// TIA Portal project "Food_Production_Automation" (V17)

(* hardware
DEVICE "HMI_1"  KTP700 Basic PN
   slot 0: "HMI_1"  KTP700 Basic PN  6AV2 123-2GB03-0AX0  17.0.0.0
   slot 1: "HMI_RT_1"  KTP700 Basic PN  6AV2 123-2GB03-0AX0  17.0.0.0
   slot 5: "HMI_1.IE_CP_1"  PROFINET Interface  17.0.0.0
      slot 1: "PROFINET Interface_1"  PROFINET Interface
         slot 1: "Port_1"  Port
DEVICE "S7-1200 station_1"  S7-1200 Station
   slot 0: "Rack_0"  S7-1200 Rack  Rack  V1.0
   slot 1: "PLC_1"  CPU 1215C DC/DC/DC  6ES7 215-1AG40-0XB0  V4.5
   slot 2: "AI 4xRTD_1"  SM 1231 AI4 x RTD  6ES7 231-5PD32-0XB0  V2.0
*)

// ===== PLC "PLC_1"  CPU 1215C DC/DC/DC =====

VAR_GLOBAL   // PLC tag table "Default tag table"
   "Tank 1 Desired Temperature" AT %MD10 : Real;
   "Tank 2 Desired Temperature" AT %MD14 : Real;
   "Tank 1 PT100 Raw" AT %IW96 : Int;
   "Tank 1 PT100 Real" AT %MD18 : Real;
   "Tank 1 Current Temperature" AT %MD22 : Real;
   "Tank 2 PT100" AT %IW98 : Int;
   "Tank 2 PT100 Real" AT %MD26 : Real;
   "Tank 2 Current Temperature" AT %MD30 : Real;
   "HMI Start Stop Button" AT %M34.0 : Bool;
   "Heater 1" AT %Q0.0 : Bool;
   "Heater 2" AT %Q0.1 : Bool;
END_VAR

ORGANIZATION_BLOCK "Main"   // OB1, LAD, ProgramCycle
TITLE = "Main Program Sweep (Cycle)"
{ S7_Optimized_Access := 'TRUE' }
VERSION : 0.1
   VAR_INPUT
      Initial_Call : Bool;   // Initial call of this OB
      Remanence : Bool;   // =True, if remanent data are available
   END_VAR
BEGIN

REGION Network 1
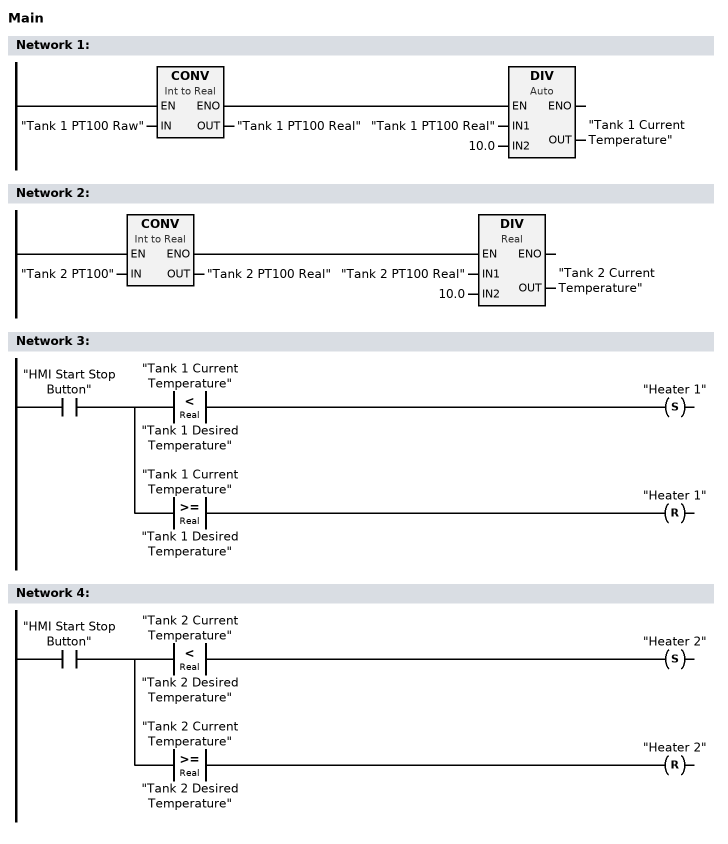
   RUNG wire#powerrail
      { S7_Templates := "[SrcType := Int, DestType := Real]" } Convert(in := "Tank 1 PT100 Raw", out => "Tank 1 PT100 Real")
      Div(in1 := "Tank 1 PT100 Real", in2 := 10.0, out => "Tank 1 Current Temperature")
   END_RUNG
   // the same network as SCL:
   "Tank 1 PT100 Real" := INT_TO_REAL("Tank 1 PT100 Raw");
   "Tank 1 Current Temperature" := "Tank 1 PT100 Real" / 10.0;
END_REGION

REGION Network 2
   RUNG wire#powerrail
      { S7_Templates := "[SrcType := Int, DestType := Real]" } Convert(in := "Tank 2 PT100", out => "Tank 2 PT100 Real")
      { S7_Templates := "SrcType := Real" } Div(in1 := "Tank 2 PT100 Real", in2 := 10.0, out => "Tank 2 Current Temperature")
   END_RUNG
   // the same network as SCL:
   "Tank 2 PT100 Real" := INT_TO_REAL("Tank 2 PT100");
   "Tank 2 Current Temperature" := "Tank 2 PT100 Real" / 10.0;
END_REGION

REGION Network 3
   RUNG wire#powerrail
      Contact( "HMI Start Stop Button" )
      wire#w1
      { S7_Templates := "SrcType := Real" } LT_Contact(in1 := "Tank 1 Current Temperature", in2 := "Tank 1 Desired Temperature")
      S_Coil( "Heater 1" )
   END_RUNG
   RUNG wire#w1
      { S7_Templates := "SrcType := Real" } GE_Contact(in1 := "Tank 1 Current Temperature", in2 := "Tank 1 Desired Temperature")
      R_Coil( "Heater 1" )
   END_RUNG
   // the same network as SCL:
   IF "HMI Start Stop Button" AND ("Tank 1 Current Temperature" < "Tank 1 Desired Temperature") THEN
       "Heater 1" := TRUE;
   END_IF;
   IF "HMI Start Stop Button" AND ("Tank 1 Current Temperature" >= "Tank 1 Desired Temperature") THEN
       "Heater 1" := FALSE;
   END_IF;
END_REGION

REGION Network 4
   RUNG wire#powerrail
      Contact( "HMI Start Stop Button" )
      wire#w1
      { S7_Templates := "SrcType := Real" } LT_Contact(in1 := "Tank 2 Current Temperature", in2 := "Tank 2 Desired Temperature")
      S_Coil( "Heater 2" )
   END_RUNG
   RUNG wire#w1
      { S7_Templates := "SrcType := Real" } GE_Contact(in1 := "Tank 2 Current Temperature", in2 := "Tank 2 Desired Temperature")
      R_Coil( "Heater 2" )
   END_RUNG
   // the same network as SCL:
   IF "HMI Start Stop Button" AND ("Tank 2 Current Temperature" < "Tank 2 Desired Temperature") THEN
       "Heater 2" := TRUE;
   END_IF;
   IF "HMI Start Stop Button" AND ("Tank 2 Current Temperature" >= "Tank 2 Desired Temperature") THEN
       "Heater 2" := FALSE;
   END_IF;
END_REGION
END_ORGANIZATION_BLOCK

(* ===== HMI "HMI_RT_1" =====
system functions are stored by id; their names below are inferred from use
connection "HMI_Connection_1": ETHERNET, SMART_S7_1200_OMS

HMI tags "Default tag table"
   "Tank 1 Desired Temperature" : Real = PLC "Tank 1 Desired Temperature" AT %MD10, 1 s
   "Tank 2 Desired Temperature" : Real = PLC "Tank 2 Desired Temperature" AT %MD14, 1 s
   "Tank 1 Current Temperature" : Real = PLC "Tank 1 Current Temperature" AT %MD22, 1 s
   "Tank 2 Current Temperature" : Real = PLC "Tank 2 Current Temperature" AT %MD30, 1 s
   "Heater 1" : Bool = PLC "Heater 1" AT %Q0.0, 1 s
   "Heater 2" : Bool = PLC "Heater 2" AT %Q0.1, 1 s
   "HMI Start Stop Button" : Bool = PLC "HMI Start Stop Button" AT %M34.0, 1 s

recipe "Recipe_1": Tank 1 Desired Temperature <- "Tank 1 Desired Temperature", Tank 2 Desired Temperature <- "Tank 2 Desired Temperature"

screen "Root screen" 800x480, template "Template_1"
   TextField "Text field_1" at 194,5 size 408x32; Text 'FOOD PRODUCTION AUTOMATION'
   GraphicView "Graphic view_3" at 84,252 size 87x48; Picture "Graphic_3"
   GraphicView "Graphic view_2" at 24,123 size 114x199; Picture "Graphic_2"
   GraphicView "Graphic view_1" at 254,252 size 87x48; Picture "Graphic_3"
   GraphicView "Graphic view_4" at 194,123 size 114x199; Picture "Graphic_2"
   GraphicView "Graphic view_5" at 48,156 size 66x67; Picture "Graphic_4"
   GraphicView "Graphic view_6" at 217,156 size 66x67; Picture "Graphic_4"
   Rectangle "Rectangle_1" at 64,240 size 30x30
      Appearance <- "Heater 1"
   Rectangle "Rectangle_2" at 235,240 size 30x30
      Appearance <- "Heater 2"
   TextField "Text field_2" at 49,294 size 61x23; Text 'Tank 1'
   TextField "Text field_3" at 219,294 size 61x23; Text 'Tank 2'
   GraphicView "Graphic view_7" at 54,319 size 50x50; Picture "Graphic_5"
   GraphicView "Graphic view_8" at 225,319 size 50x50; Picture "Graphic_6"
   GraphicView "Graphic view_9" at 102,319 size 126x50; Picture "Graphic_7"
   GraphicView "Graphic view_10" at 271,319 size 126x50; Picture "Graphic_7"
   GraphicView "Graphic view_11" at 393,319 size 50x50; Picture "Graphic_8"
   IOField "I/O field_1" at 50,94 size 63x28; FormatPattern 99.9
      ProcessValue <- "Tank 1 Current Temperature"
   TextField "Text field_4" at 6,74 size 154x18; Text 'CURRENT TEMPERATURE'
   IOField "I/O field_2" at 218,94 size 63x28; FormatPattern 99.9
      ProcessValue <- "Tank 2 Current Temperature"
   TextField "Text field_5" at 174,74 size 154x18; Text 'CURRENT TEMPERATURE'
   TextField "Text field_6" at 280,96 size 24x23; Text '°C'
   TextField "Text field_7" at 112,97 size 24x23; Text '°C'
   IOField "I/O field_3" at 48,385 size 63x28; FormatPattern 99
      ProcessValue <- "Tank 1 Desired Temperature"
   TextField "Text field_8" at 5,365 size 152x18; Text 'DESIRED TEMPERATURE'
   TextField "Text field_9" at 111,388 size 24x23; Text '°C'
   IOField "I/O field_4" at 219,385 size 63x28; FormatPattern 99
      ProcessValue <- "Tank 2 Desired Temperature"
   TextField "Text field_10" at 176,365 size 152x18; Text 'DESIRED TEMPERATURE'
   TextField "Text field_11" at 282,388 size 24x23; Text '°C'
   Button "Button_1" at 113,435 size 96x32; TextOff 'ON/OFF'
      on Press: InvertBit("HMI Start Stop Button")
   RecipeView "Recipe view_1" at 446,73 size 347x401; DataRecordNameCaption 'Product Name:'; EntryNameCaption 'Liquid Temperature'; Recipe "Recipe_1"
*)